{attribute addProperty BoxType "EM7004-0000-0016"}
{attribute addProperty Id "Latch_extern_validAT %I*BOOL812Set_counter_doneAT %I*BOOL813Status_of_input_AAT %I*BOOL819Status_of_input_BAT %I*BOOL8110Status_of_input_gateAT %I*BOOL8112Status_of_extern_latchAT %I*BOOL8113TxPDO_ToggleAT %I*BOOL819Counter_valueAT %I*UINT16217Latch_valueAT %I*UINT16218"}
{attribute addProperty CRC "2409141999"}
{attribute addProperty SizeInBites "88"}
{attribute addProperty SizeInBytes "11"}
TYPE ENC_Inputs_Channel_8F9896EF :
STRUCT
	{attribute addProperty Name "Latch_extern_valid"}
	Latch_extern_valid AT %I* : BOOL;
	{attribute addProperty Name "Set_counter_done"}
	Set_counter_done AT %I* : BOOL;
	{attribute addProperty Name "Status_of_input_A"}
	Status_of_input_A AT %I* : BOOL;
	{attribute addProperty Name "Status_of_input_B"}
	Status_of_input_B AT %I* : BOOL;
	{attribute addProperty Name "Status_of_input_gate"}
	Status_of_input_gate AT %I* : BOOL;
	{attribute addProperty Name "Status_of_extern_latch"}
	Status_of_extern_latch AT %I* : BOOL;
	{attribute addProperty Name "TxPDO_Toggle"}
	TxPDO_Toggle AT %I* : BOOL;
	{attribute addProperty Name "Counter_value"}
	Counter_value AT %I* : UINT;
	{attribute addProperty Name "Latch_value"}
	Latch_value AT %I* : UINT;
END_STRUCT
END_TYPE

(* stored: Version 1.2.0.0, ProductVersion 3.1.4024.9
   DUT ENC_Inputs_Channel_8F9896EF: Id {8f4a18db-b0ac-4dcc-90fd-37083671e427} *)
